{attribute 'GeneratedUsingTerminal: EL5001-0011-0019'}
{attribute addProperty BoxType "EL5001-0011-0019"}
{attribute addProperty Id "StatusAT %I*Status_536663CA5Counter_valueAT %I*UDINT4"}
{attribute addProperty CRC "2344717740"}
{attribute addProperty Size "9"}
TYPE SSI_Inputs_8BC18DAC :
STRUCT
	{attribute addProperty Name "Status"}
	Status AT %I* : Status_536663CA;
	{attribute addProperty Name "Counter_value"}
	Counter_value AT %I* : UDINT;
END_STRUCT
END_TYPE

(* stored: Version 1.2.0.0, ProductVersion 3.1.4024.9
   DUT SSI_Inputs_8BC18DAC: Id {5880ed8f-6a6c-4559-a944-dcb2f1fdf67e} *)
